// TIA Portal V19 export
FUNCTION "M_PosAMinusCostB" : LReal   // FC26, LAD
TITLE = Module POSA minus CostantB / Position A minus Costant B
// stored: Access Published, SetENOAutomatically false
   VAR_INPUT
      PosA : LReal;
      CostB : LReal;
      MODULE : LReal;
   END_VAR
   VAR_TEMP
      Xc : LReal;
   END_VAR
BEGIN

REGION Network 1 (SCL): Xc = PosA - CostB / Main
   #Xc := #PosA - #CostB;
   #M_PosAMinusCostB := #Xc;

   IF #MODULE > 0.0 THEN
       IF #Xc >= #MODULE THEN
           #M_PosAMinusCostB := #Xc - #MODULE;
       ELSIF #Xc < 0 THEN
           #M_PosAMinusCostB := #MODULE + #Xc;
       END_IF;
       IF ABS(#M_PosAMinusCostB - #MODULE) < 0.01 THEN
           #M_PosAMinusCostB := 0;
       END_IF;
   END_IF;
END_REGION
END_FUNCTION
